// TIA Portal V16 export
// export: Created 2021-08-04T22:56:06.6957166Z, ExportSetting WithDefaults, DisplayName Totally Integrated Automation Portal, DisplayVersion V16 Update 4, DisplayName TIA Portal Version Control Interface, DisplayVersion V16 Update 2, DisplayName TIA Portal Openness, DisplayVersion V16 Update 4, DisplayName STEP 7 Professional, DisplayVersion V16 Update 4, DisplayName STEP 7 Safety, DisplayVersion V16, DisplayName WinCC Advanced, DisplayVersion V16 Update 4
FUNCTION_BLOCK "MyCounter"   // FB2, F_FBD
{ S7_Optimized_Access := 'TRUE' }
VERSION : 0.1
// stored: AutoNumber true, IsIECCheckEnabled false, UDAEnableTagReadback false
   VAR_INPUT
      increment : Int;
   END_VAR
   VAR
      "counter" : Int;
   END_VAR
BEGIN

REGION Network 1
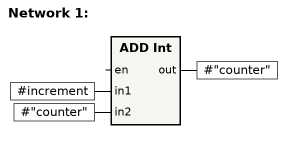
   #"counter" := #increment + #"counter";
END_REGION
END_FUNCTION_BLOCK
